Staubli VAL3: iIdent2.pgx

public program iIdent2(num& nNum[] (dimensions=1))
begin
  nNum=dioGet(iIdent2)
end
